// POUs/StringHelper/getCntCharInStr
{attribute 'no_check'}
//Returns the count of a particular char found in a string line
FUNCTION getCntCharInStr : INT
VAR_INPUT
	Chars													:	STRING(5):=';';
	Strline													:	T_MaxString;
END_VAR             										
VAR                 
	tmpString												:	T_MaxString ;										
	pos,k													:	INT;
END_VAR

IF StrLine <> '' AND Chars <> ''
THEN
	MEMSET(ADR(tmpString),0,SIZEOF(tmpString));
	MEMCPY(ADR(tmpString),ADR(Strline),TO_UDINT(LEN(Strline)));
	pos 													:= FIND (tmpString,Chars);
	WHILE pos <> 0 DO	
		k													:=  pos + (LEN(Chars) - 1);
		tmpString											:=	RIGHT(tmpString,LEN(tmpString) - k);
		pos 												:= 	FIND (tmpString,Chars);
		getCntCharInStr										:=	getCntCharInStr+1;
	END_WHILE;
ELSE
	getCntCharInStr											:= 0;
END_IF

END_FUNCTION

// POUs/StringHelper/getCntCharInWStr
{attribute 'no_check'}
//Returns the count of a particular char found in a string line
FUNCTION getCntCharInWStr : INT
VAR_INPUT
	Char													:	WSTRING(3):=";";
	Strline													:	WSTRING(MAX_STRING_LENGTH);
END_VAR             										
VAR                 
	tmpString												:	WSTRING(MAX_STRING_LENGTH) ;										
	pos,k													:	INT;
END_VAR

IF Strline <> "" AND Char <> ""
THEN	
	MEMSET(ADR(tmpString),0,SIZEOF(tmpString));
	MEMCPY(ADR(tmpString),ADR(Strline),TO_UDINT(WLEN(Strline) * 2));
	pos 													:= WFIND (tmpString,char);
	WHILE pos <> 0 DO		
		k													:=  pos + (WLEN(char) - 1);
		tmpString											:=	WRIGHT(tmpString,WLEN(tmpString) - k);
		pos 												:= 	WFIND (tmpString,char);
		getCntCharInWStr									:=	getCntCharInWStr+1;
	END_WHILE;
ELSE
	getCntCharInWStr										:= 0;
END_IF

END_FUNCTION

// POUs/StringHelper/getFilledString
{attribute 'no_check'}
//Returns a string which is filled with a defined char on the left or right site with a desired lenght  
FUNCTION getFilledString : T_MaxString
VAR_INPUT
	Strline													:	T_MaxString;	//Start string
	Lenght													:	INT;			//Desired lenght
	FillChar												:	STRING(1);		//Fill char
	LeftInsert												:	BOOL;			//Insert char on left site of start string
END_VAR             										
VAR                 										
	tmp														:	T_MaxString;
	i 														: INT;
END_VAR

GetFilledString 											:= Strline;
tmp 														:= '';

FOR i := 0 TO Lenght DO
	IF LEN(getFilledString)+ Lenght >= UINT_TO_INT(SIZEOF(getFilledString)) 
	THEN
		RETURN;
	ELSE
		IF LeftInsert 
		THEN
			IF LEN(tmp) < Lenght - LEN(Strline) 
			THEN
				tmp 										:= INSERT(tmp,FillChar,LEN(tmp));
			ELSE
				getFilledString 							:= CONCAT(tmp,getFilledString);
			END_IF                  						
		ELSE                        						
			getFilledString									:= INSERT(getFilledString,FillChar,LEN(getFilledString));
		END_IF
	END_IF
END_FOR

END_FUNCTION

// POUs/StringHelper/HEXSTR_TO_DWORD
{attribute 'no_check'}
//Converts a hex string into a 32 bit DWORD number
FUNCTION HEXSTR_TO_DWORD : BOOL //Return value TRUE = successful converted / FALSE if there are no valid hex signs or seperators
VAR_INPUT
	Hexstring 												: T_MaxString;
END_VAR
VAR_IN_OUT
{attribute 'displaymode':='hexadecimal'}
	Target													: DWORD;
END_VAR
VAR
	HexMarkerFound											: BOOL;
	i,j,Max_i,Max_j											: INT;
{attribute 'displaymode':='hexadecimal'}
	X														: BYTE;
{attribute 'displaymode':='hexadecimal'}
	TmpTarget												: DWORD;
END_VAR

Max_i 														:= LEN(Hexstring) - 1;
Max_j														:= SIZEOF(Target) * 2;
TmpTarget													:= 0;
HEXSTR_TO_DWORD												:= TRUE;
FOR i := 0 TO Max_i DO
	(* read the first character and subtract 48 to get value in decimal 0 = 48 *)
	(* calculate the value of the digit *)
	X														:= Hexstring[i];
	IF j >= Max_j
	THEN
		EXIT;
	ELSIF X > 47 AND x < 58 
	THEN //x = number 0-9
		TmpTarget 											:= SHL(TmpTarget,4) + X - 48;
		j													:= j + 1;
	ELSIF X > 64 AND X < 71 								
	THEN //x = letter A-F                   								
		TmpTarget 											:= SHL(TmpTarget,4) + X - 55;
		j													:= j + 1;
	ELSIF X > 96 AND X < 103								 
	THEN //x = letter a-f                     								
		TmpTarget 											:= SHL(TmpTarget,4) + X - 87;
		j													:= j + 1;
	ELSIF x = 16#58 OR x = 16#78 OR  x = 16#23
	THEN //found x, X or #, start over again because of 0xFA or 16#AB
		IF HexMarkerFound
		THEN
			HEXSTR_TO_DWORD									:= FALSE;	
			RETURN;		
		ELSE
			TmpTarget										:= 0;
			HexMarkerFound									:= TRUE;
			j												:= 0;	
		END_IF		
	ELSIF X = 16#2C OR X = 16#3A OR X = 16#2E OR X = 16#3B OR X = 16#20 OR X = 16#5F
	THEN //Ignore comma,colon,dot,space,underline
		; 
	ELSE
		HEXSTR_TO_DWORD										:= FALSE;	
		RETURN;
	END_IF
END_FOR
Target														:= TmpTarget;

END_FUNCTION

// POUs/StringHelper/HEXSTR_TO_LWORD
{attribute 'no_check'}
//Converts a hex string into a 64 bit LWORD number
FUNCTION HEXSTR_TO_LWORD : BOOL //Return value TRUE = successful converted / FALSE if there are no valid hex signs or seperators
VAR_INPUT
	Hexstring 												: T_MaxString;
END_VAR
VAR_IN_OUT
{attribute 'displaymode':='hexadecimal'}
	Target													: LWORD;
END_VAR
VAR
	HexMarkerFound											: BOOL;
	i,j,Max_i,Max_j											: INT;
{attribute 'displaymode':='hexadecimal'}
	X														: BYTE;
{attribute 'displaymode':='hexadecimal'}
	TmpTarget												: LWORD;
END_VAR

Max_i 														:= LEN(Hexstring) - 1;
Max_j														:= SIZEOF(Target) * 2;
TmpTarget 													:= 0;
HEXSTR_TO_LWORD												:= TRUE;
FOR i := 0 TO Max_i DO
	(* read the first character and subtract 48 to get value in decimal 0 = 48 *)
	(* calculate the value of the digit *)
	X														:= Hexstring[i];
	IF j >= Max_j
	THEN
		EXIT;
	ELSIF X > 47 AND x < 58 
	THEN //x = number 0-9
		TmpTarget 											:= SHL(TmpTarget,4) + X - 48;
		j													:= j + 1;
	ELSIF X > 64 AND X < 71 								
	THEN //x = letter A-F                   								
		TmpTarget 											:= SHL(TmpTarget,4) + X - 55;
		j													:= j + 1;
	ELSIF X > 96 AND X < 103								 
	THEN //x = letter a-f                     								
		TmpTarget 											:= SHL(TmpTarget,4) + X - 87;
		j													:= j + 1;
	ELSIF x = 16#58 OR x = 16#78 OR  x = 16#23
	THEN //found x, X or #, start over again because of 0xFA or 16#AB
		IF HexMarkerFound
		THEN
			HEXSTR_TO_LWORD									:= FALSE;	
			RETURN;		
		ELSE
			TmpTarget										:= 0;
			HexMarkerFound									:= TRUE;
			j												:= 0;	
		END_IF		
	ELSIF X = 16#2C OR X = 16#3A OR X = 16#2E OR X = 16#3B OR X = 16#20 OR X = 16#5F
	THEN //Ignore comma,colon,dot,space,underline
		; 
	ELSE
		HEXSTR_TO_LWORD										:= FALSE;	
		RETURN;
	END_IF
END_FOR
Target														:= TmpTarget;

END_FUNCTION

// POUs/StringHelper/isWStringNumeric
{attribute 'no_check'}
//Returns TRUE in case a ascii string contains only a valid number signs. Minus,plus,space,comma and dot are allowed
//Limited to a Param.MAX_EXT_STRING_LENGTH long string  
FUNCTION isWStringNumeric : BOOL 
VAR_INPUT
	pSource													:	POINTER TO WORD;
END_VAR             										
VAR                 
	Cr														:	WORD;	//Char									
	countSeperator											:	INT;
	i														:	UDINT;
	Addr													:	POINTER TO WORD;
END_VAR

IF pSource <> 0
THEN
	isWStringNumeric										:=	TRUE;
	FOR i := 0 TO PARAM.MAX_EXT_STRING_LENGTH DO
		Addr												:= pSource + (i * 2);
		Cr												:= Addr^;
		IF Cr = 0
		THEN 														
			isWStringNumeric								:= i > 0; //Only TRUE if string is not empty 
			EXIT;
		ELSIF Cr = 46 OR Cr = 44 //comma or point as a seperator
		THEN
			countSeperator									:= countSeperator + 1;
			IF countSeperator > 1 
			THEN
				isWStringNumeric							:= FALSE;
				EXIT;	(* more than one seperator -> no number *)
			END_IF
		ELSIF(Cr < 48 OR Cr > 57)
			AND Cr <> 45 (* minus *)
			AND Cr <> 43 (* plus *)
			AND Cr <> 32 (* Space *)
			AND Cr <> 101(* e for 9.9999992e-2 *)
			OR i = PARAM.MAX_EXT_STRING_LENGTH
		THEN
			isWStringNumeric								:= FALSE;
			EXIT;	(* no numerical char *)
		END_IF
	END_FOR      
ELSE
	isWStringNumeric										:= FALSE;
END_IF

END_FUNCTION

// POUs/StringHelper/LWORD_TO_BINSTR_EXT
{attribute 'no_check' := ''}
FUNCTION LWORD_TO_BINSTR_EXT : T_MaxString //This function converts a decimal number into a binary string (base 2), where the digits are separated according to the selected mode 
//e.g. 1111000011110000 -> 1111_0000_1111_0000 
VAR_INPUT
	In														: LWORD;//The decimal number requiring conversion.
	Precision												: INT; //Minimum number of displayed digits (digits), filled up with 0 from left if significant digits are less then that
	Mode													: INT; //1=Separate high and low word / 2=Separate bytes / 3=Separate nibbles /ELSE no separation | Separator = Param.DOWRD_TO_XXXSTR_EXT_SEPARATOR
END_VAR
VAR													
END_VAR

LWORD_TO_BINSTR_EXT 										:= LWORD_TO_BINSTR(in,precision);

CASE mode OF
1:// Separate by low word and high word
	LWORD_TO_BINSTR_EXT										:= INSERT_EXT(LWORD_TO_BINSTR_EXT,PARAM.XWORD_TO_XXXSTR_EXT_SEPARATOR,16);
	
2://Separate by bytes
	LWORD_TO_BINSTR_EXT										:= INSERT_EXT(LWORD_TO_BINSTR_EXT,PARAM.XWORD_TO_XXXSTR_EXT_SEPARATOR,8);
	
3://Separate by nibble
	LWORD_TO_BINSTR_EXT										:= INSERT_EXT(LWORD_TO_BINSTR_EXT,PARAM.XWORD_TO_XXXSTR_EXT_SEPARATOR,4);
END_CASE

END_FUNCTION

// POUs/StringHelper/LWORD_TO_HEXSTR_EXT
{attribute 'no_check' := ''}
FUNCTION LWORD_TO_HEXSTR_EXT : T_MaxString //This function converts a decimal number into a hexadecimal string (base 16)., where the hex signs are separated according to the selected mode 
//e.g. F0F0F0F0 -> F0_F0_F0_F0 
VAR_INPUT
	In														: LWORD;
	Precision												: INT;//Minimum number of displayed signs, filled up with 0 from left if significant digits are less then that
	LoCase													: BOOL;
	Mode													: INT; //1=parted by word, 2=parted by byte, 3=parted by nibble
END_VAR
VAR
END_VAR

LWORD_TO_HEXSTR_EXT 										:= LWORD_TO_HEXSTR(in,precision,loCase);
CASE mode OF
1:// Separate by low word and high word
	LWORD_TO_HEXSTR_EXT										:= INSERT_EXT(LWORD_TO_HEXSTR_EXT,PARAM.XWORD_TO_XXXSTR_EXT_SEPARATOR,4);
	
2://Separate by bytes
	LWORD_TO_HEXSTR_EXT										:= INSERT_EXT(LWORD_TO_HEXSTR_EXT,PARAM.XWORD_TO_XXXSTR_EXT_SEPARATOR,2);
	
3://Separate by nibble
	LWORD_TO_HEXSTR_EXT										:= INSERT_EXT(LWORD_TO_HEXSTR_EXT,PARAM.XWORD_TO_XXXSTR_EXT_SEPARATOR,1);
END_CASE

END_FUNCTION

// POUs/StringHelper/readWStrToSeperator
{attribute 'no_check'}
//Returns a wstring found on the left side of a seperator, empty if seperator is not found
FUNCTION readWStrToSeperator : WSTRING(MAX_STRING_LENGTH)
VAR_INPUT
	Seperator												:	WSTRING(10) :=";";
	Strline													:	WSTRING(MAX_STRING_LENGTH);
END_VAR
VAR_IN_OUT
END_VAR
VAR
	pos														:	INT;
END_VAR

IF strline = ""
THEN
	readWStrToSeperator										:= "";
ELSE
	pos 													:= WFIND (strline,seperator);
	IF (pos >= 1) 
	THEN
		readWStrToSeperator									:= WLEFT (strline,pos-1);
	ELSE
		readWStrToSeperator									:= "";
	END_IF
END_IF

END_FUNCTION

// POUs/StringHelper/replaceInString
{attribute 'no_check'}
//Replace a part of a string with another string 
FUNCTION replaceInString : BOOL
VAR_INPUT
	SearchStr												:	STRING(10); //e.g. '/r/n_
	ReplaceStr												:	STRING(10); //e.g. '-'
END_VAR             										
VAR_IN_OUT         										
	Strline													: 	T_MaxString;
END_VAR             										
VAR                 	
	StrLen, i,pos											:	INT;
END_VAR

IF strline = '' 
THEN 
	replaceInString											:= TRUE;
ELSE
	StrLen													:= LEN(strline);
	FOR i := 0 TO StrLen
	DO
		pos 												:= FIND(strline,SearchStr);
		IF pos >= 1 
		THEN
			strline											:= REPLACE(strline,ReplaceStr,LEN(SearchStr),pos);
		ELSE
			replaceInString									:= i > 0; 
			EXIT;						
		END_IF	
	END_FOR
END_IF

END_FUNCTION

// POUs/StringHelper/replaceInWString
{attribute 'no_check'}
//Replace a part of a string with another string 
FUNCTION replaceInWString : BOOL
VAR_INPUT
	SearchStr												:	WSTRING(10); //e.g. '/r/n_
	ReplaceStr												:	WSTRING(10); //e.g. '-'
END_VAR             										
VAR_IN_OUT         										
	Strline													: 	WSTRING(MAX_STRING_LENGTH);
END_VAR             										
VAR                 	
	StrLen, i,pos											:	INT;
END_VAR

IF strline = "" 
THEN 
	replaceInWString										:= TRUE;
ELSE
	StrLen													:= WLEN(strline);
	FOR i := 0 TO StrLen
	DO
		pos 												:= WFIND(strline,SearchStr);
		IF pos >= 1 
		THEN
			strline											:= WREPLACE(strline,ReplaceStr,WLEN(SearchStr),pos);
		ELSE
			replaceInWString								:= i > 0; 
			EXIT;						
		END_IF	
	END_FOR
END_IF

END_FUNCTION

// POUs/StringHelper/replaceUmlauts
// ReplaceUmlauts replaces all "german" umlauts in an given string Ä-> ae | ä -> ae | Ö -> oe | ö -> oe | Ü -> ue | ü -> ue | ß -> ss 
FUNCTION replaceUmlauts : INT // returns no of replaced umlauts
VAR_IN_OUT
	SearchStr		: T_MaxString;				
END_VAR
VAR
	i			: INT;
END_VAR

FOR i := 0 TO LEN(SearchStr) DO
	CASE SearchStr[i] OF
	196:	// Ä
		SearchStr 					:= REPLACE(SearchStr, 'Ae', 1, i+1); 
		i 							:= i + 1;
		ReplaceUmlauts 				:= ReplaceUmlauts + 1;
	214:	// Ö
		SearchStr 					:= REPLACE(SearchStr, 'Oe', 1, i+1);
		i 							:= i + 1; 
		ReplaceUmlauts 				:= ReplaceUmlauts + 1;
	220:	// Ü
		SearchStr 					:= REPLACE(SearchStr, 'Ue', 1, i+1);
		i 							:= i + 1; 
		ReplaceUmlauts 				:= ReplaceUmlauts + 1;
	223:	// ß
		SearchStr 					:= REPLACE(SearchStr, 'ss', 1, i+1);
		i 							:= i + 1; 
		ReplaceUmlauts 				:= ReplaceUmlauts + 1;	
	228:	// ä
		SearchStr 					:= REPLACE(SearchStr, 'ae', 1, i+1);
		i 							:= i + 1; 
		ReplaceUmlauts 				:= ReplaceUmlauts + 1;
	246:	// ö
		SearchStr 					:= REPLACE(SearchStr, 'oe', 1, i+1);
		i 							:= i + 1; 
		ReplaceUmlauts 				:= ReplaceUmlauts + 1;
	252:	// ü
		SearchStr 					:= REPLACE(SearchStr, 'ue', 1, i+1);
		i 							:= i + 1; 
		ReplaceUmlauts 				:= ReplaceUmlauts + 1;
	ELSE	// nothing replaced in this cycle	
		;
	END_CASE
END_FOR

END_FUNCTION

// POUs/StringHelper/WINSERT_EXT
{attribute 'no_check' := ''}
FUNCTION WINSERT_EXT : WSTRING //The function WINSERT_EXT inserts WSTR2 into WSTR1 at every ITERATION_POSs position  
VAR_INPUT
	STR1													:WSTRING; //Base string - Hint! The base string will cut off if iteration of insertions exceeded the size of the string variable 
	STR2													:WSTRING; //Insert string 
	ITERATION_POS											: INT; //Insert iteration position 
END_VAR
VAR
	Length1,length2,i,iEnd									: INT;														
END_VAR

WINSERT_EXT													:= STR1;
Length1														:= WLEN(STR1);
Length2														:= WLEN(STR2);
IF TO_UINT(Length1 + Length2) > SIZEOF(STR1)
	OR ITERATION_POS = 0
THEN
	;
ELSE
	iEnd													:= ABS(Length1 / ITERATION_POS) - 1;
	FOR i := 1 TO iEnd
	DO 
		WINSERT_EXT											:= WINSERT(WINSERT_EXT,STR2,Length1 - ITERATION_POS * i);
	END_FOR
END_IF

END_FUNCTION

// POUs/System/SystemPulses
{attribute 'no_check'}
//Provides various puslse signals as default
FUNCTION_BLOCK SystemPulses
VAR_INPUT
{attribute 'displaymode':='binary'}
	Options													:	WORD := 2#0000_0001_1110_1110; //Set bit in Options word to enable ot disable existing pulse instances
	PT_ON_Custom											:	TIME := T#30S;	
	PT_OFF_Custom											:	TIME := T#30S;
END_VAR
VAR_OUTPUT
	BlinkSlow												: 	BOOL;
	Blink													: 	BOOL;
	BlinkFast												: 	BOOL;
	BlinkVeryFast											:	BOOL;
	BlinkFlash												:	BOOL;
	
	_20ms													: 	Pulse := (IN := TRUE,	PT_OFF := T#20MS, 		PT_ON := T#20MS);	//20ms						Options .0
	_100ms													: 	Pulse := (IN := TRUE,	PT_OFF := T#100MS, 		PT_ON := T#100MS); 	//10Hz (0.1s) pulse			Options .1
	_250ms													: 	Pulse := (IN := TRUE,	PT_OFF := T#250MS, 		PT_ON := T#250MS); 	//4 Hz - Blink very Fast	Options .2
	_400ms													: 	Pulse := (IN := TRUE,	PT_OFF := T#400MS, 		PT_ON := T#400MS); 	//2.5Hz - Blink Fast *)		Options .3
	_500ms													: 	Pulse := (IN := TRUE,	PT_OFF := T#500MS, 		PT_ON := T#500MS); 	//2Hz / 500ms				Options .4
	_800ms													: 	Pulse := (IN := TRUE,	PT_OFF := T#800MS, 		PT_ON := T#800MS); 	//1.25Hz - Blink normal 	Options .5
	_1s														: 	Pulse := (IN := TRUE,	PT_OFF := T#1S, 		PT_ON := T#1S); 	//1Hz /1s					Options .6
	_1s600ms												: 	Pulse := (IN := TRUE,	PT_OFF := T#1S600MS, 	PT_ON := T#1S600MS);//0.625Hz - Blink slow 		Options .7
	_2s														: 	Pulse := (IN := TRUE,	PT_OFF := T#2S, 		PT_ON := T#2S); 	//0.5Hz						Options .8
	_5s														: 	Pulse := (IN := TRUE,	PT_OFF := T#5S, 		PT_ON := T#5S); 	//5s						Options .9
	_10s													: 	Pulse := (IN := TRUE, 	PT_OFF := T#10S, 		PT_ON := T#10S); 	//10s						Options .10
	_1m														: 	Pulse := (IN := TRUE, 	PT_OFF := T#1M, 		PT_ON := T#1M); 	//1m						Options .11	
	_5m														: 	Pulse := (IN := TRUE, 	PT_OFF := T#5M, 		PT_ON := T#5M); 	//5m						Options .12
	_10m													: 	Pulse := (IN := TRUE, 	PT_OFF := T#10M, 		PT_ON := T#10M); 	//10m						Options .13
	_60m													: 	Pulse := (IN := TRUE, 	PT_OFF := T#60M, 		PT_ON := T#60M); 	//60m						Options .14
	_Custom													: 	Pulse := (IN := TRUE, 	PT_OFF := T#30S, 		PT_ON := T#60M); 	//60m						Options .15
	_Flash													: 	Pulse := (IN := TRUE, 	PT_OFF := T#800MS, 		PT_ON := T#80MS);	//800ms/80ms Blink as flash light
END_VAR                                                            
VAR                                                                
END_VAR

(************************************************************************************************************)
(* function-block generates different pulse signals															*)
(************************************************************************************************************)

(* impuls generator *****************************************************************************************)
_Flash(Q => BlinkFlash); 
IF Options.0 THEN _20ms(Q => ); 				END_IF
IF Options.1 THEN _100ms(Q => ); 				END_IF
IF Options.2 THEN _250ms(Q => BlinkVeryFast); 	END_IF
IF Options.3 THEN _400ms(Q => BlinkFast); 		END_IF
IF Options.4 THEN _500ms(Q => ); 				END_IF
IF Options.5 THEN _800ms(Q => Blink); 			END_IF
IF Options.6 THEN _1s(Q => ); 					END_IF
IF Options.7 THEN _1s600ms(Q => BlinkSlow); 	END_IF
IF Options.8 THEN _2s(Q => ); 					END_IF
IF Options.9 THEN _5s(Q => ); 					END_IF
IF Options.10 THEN _10s(Q => ); 				END_IF
IF Options.11 THEN _1m(Q => ); 					END_IF
IF Options.12 THEN _5m(Q => ); 					END_IF
IF Options.13 THEN _10m(Q => ); 				END_IF
IF Options.14 THEN _60m(Q => ); 				END_IF
IF Options.15 THEN _Custom(PT_OFF := PT_OFF_Custom, PT_ON := PT_ON_Custom ,Q => );	END_IF

(************************************************************************************************)

PROPERTY PUBLIC optAllOn : bool
GET
optAllOn := OPtions = 2#1111_1111_1111_1111;
END_GET
SET
If optAllOn then OPtions := 2#1111_1111_1111_1111; End_if
END_SET
END_PROPERTY

PROPERTY PUBLIC optEnable100ms : bool
GET
optEnable100ms := Options.0;
END_GET
SET
Options.0 := optEnable100ms;
END_SET
END_PROPERTY

PROPERTY PUBLIC optEnable10m : bool
GET
optEnable10m := Options.13;
END_GET
SET
Options.13 := optEnable10m;
END_SET
END_PROPERTY

PROPERTY PUBLIC optEnable10s : bool
GET
optEnable10s := Options.10;
END_GET
SET
Options.10 := optEnable10s;
END_SET
END_PROPERTY

PROPERTY PUBLIC optEnable1m : bool
GET
optEnable1m := Options.11;
END_GET
SET
Options.11 := optEnable1m;
END_SET
END_PROPERTY

PROPERTY PUBLIC optEnable1s : bool
GET
optEnable1s := Options.6;
END_GET
SET
Options.6 := optEnable1s;
END_SET
END_PROPERTY

PROPERTY PUBLIC optEnable1s600msBlinkSlow : bool
GET
optEnable1s600msBlinkSlow := Options.7;
END_GET
SET
Options.7 := optEnable1s600msBlinkSlow;
END_SET
END_PROPERTY

PROPERTY PUBLIC optEnable20ms : bool
GET
optEnable20ms := Options.0;
END_GET
SET
Options.0 := optEnable20ms;
END_SET
END_PROPERTY

PROPERTY PUBLIC optEnable250msBlinkVeryFast : bool
GET
optEnable250msBlinkVeryFast := Options.2;
END_GET
SET
Options.2 := optEnable250msBlinkVeryFast;
END_SET
END_PROPERTY

PROPERTY PUBLIC optEnable2s : bool
GET
optEnable2s := Options.8;
END_GET
SET
Options.8 := optEnable2s;
END_SET
END_PROPERTY

PROPERTY PUBLIC optEnable400msBlinkFast : bool
GET
optEnable400msBlinkFast := Options.3;
END_GET
SET
Options.3 := optEnable400msBlinkFast;
END_SET
END_PROPERTY

PROPERTY PUBLIC optEnable500ms : bool
GET
optEnable500ms := Options.4;
END_GET
SET
Options.4 := optEnable500ms;
END_SET
END_PROPERTY

PROPERTY PUBLIC optEnable5m : bool
GET
optEnable5m := Options.12;
END_GET
SET
Options.12 := optEnable5m;
END_SET
END_PROPERTY

PROPERTY PUBLIC optEnable5s : bool
GET
optEnable5s := Options.9;
END_GET
SET
Options.9 := optEnable5s;
END_SET
END_PROPERTY

PROPERTY PUBLIC optEnable60m : bool
GET
optEnable60m := Options.14;
END_GET
SET
Options.14 := optEnable60m;
END_SET
END_PROPERTY

PROPERTY PUBLIC optEnable800msBlink : bool
GET
optEnable800msBlink := Options.5;
END_GET
SET
Options.5 := optEnable800msBlink;
END_SET
END_PROPERTY

PROPERTY PUBLIC optEnableCustom : bool
GET
optEnableCustom:= Options.15;
END_GET
SET
Options.15 := optEnableCustom;
END_SET
END_PROPERTY

END_FUNCTION_BLOCK

// POUs/System/TaskInfo
{attribute 'no_check'}
//Provides all information of PlcTaskSystemInfo corresponding to the caller task of the instance 
FUNCTION_BLOCK TaskInfo
VAR_INPUT
END_VAR
VAR_OUTPUT
	Index													:	INT := 0;
	TaskName          										: 	STRING(63);
	ObjId             										: 	OTCID;
	CycleTime         										: 	UDINT;
	CycleTimeT       										: 	TIME;
	CycleTimeLT       										: 	LTIME;
	CycleTimeFloat											:	LREAL;	
	Priority          										: 	UINT;
	AdsPort           										: 	UINT;
	CycleCount        										: 	UDINT;
	Tasktime												:	ULINT;
	DcTaskTime        										: 	T_DCTIME64;
	LastExecTime      										: 	UDINT; 
	LastExecTimeNS      									: 	UDINT; //Converted in ns 
	LastExecTimeLT      									: 	LTIME; 
	MaxExecTimeLT											:	LTIME;
	FirstCycle        										: 	BOOL;
	CycleTimeExceeded 										: 	BOOL;	
	CycleTimeExceededCount 									: 	UDINT; //Set to 0 via method resetCylceTimeExceeded()
	CycleTimeExceededCountTotal 							: 	UDINT; //Overall count cycle time exeeded
	InCallAfterOutputUpdate									:	BOOL;
	RTViolation												:	BOOL;
END_VAR

VAR
	GETCURTASKINDEX											: 	GETCURTASKINDEX;
	GETTASKTIME												:	GETTASKTIME;
	TaskInterlock											:	BOOL;
END_VAR

	(*	evaluate PlcTaskInfo arrays													*)
	(********************************************************************************)

(* read task info array of caller task ************************************************************************)
	IF GETCURTASKINDEX.index = 0 	
	THEN 
		GETCURTASKINDEX(index => index); 
		//Init
		TaskName          									:= TwinCAT_SystemInfoVarList._TaskInfo[index].TaskName;
		ObjId             									:= TwinCAT_SystemInfoVarList._TaskInfo[index].ObjId;
		CycleTime         									:= TwinCAT_SystemInfoVarList._TaskInfo[index].CycleTime;
		Priority          									:= TwinCAT_SystemInfoVarList._TaskInfo[index].Priority;
		AdsPort           									:= TwinCAT_SystemInfoVarList._TaskInfo[index].AdsPort;
		CycleTimeT											:= LREAL_TO_TIME(UDINT_TO_LREAL(CycleTime) * 0.0001 );
		CycleTimeLT											:= TO_LTIME(CycleTime * 100);
		CycleTimeFloat										:= (UDINT_TO_LREAL(CycleTime) * 0.0001 / 1000.0);		
	END_IF

	//Cylic 
	CycleCount        										:= TwinCAT_SystemInfoVarList._TaskInfo[index].CycleCount;
	DcTaskTime        										:= TO_ULINT(TwinCAT_SystemInfoVarList._TaskInfo[index].DcTaskTime); 
	LastExecTime      										:= TwinCAT_SystemInfoVarList._TaskInfo[index].LastExecTime; 
	LastExecTimeNS											:= TwinCAT_SystemInfoVarList._TaskInfo[index].LastExecTime * 100;
	LastExecTimeLT      									:= TO_LTIME(LastExecTimeNS); //Converted into ns 
	MaxExecTimeLT											:= MAX(LastExecTimeLT,MaxExecTimeLT);
	
	FirstCycle        										:= TwinCAT_SystemInfoVarList._TaskInfo[index].FirstCycle;
	CycleTimeExceeded 										:= TwinCAT_SystemInfoVarList._TaskInfo[index].CycleTimeExceeded;
	IF CycleTimeExceeded 
	THEN
		CycleTimeExceededCount								:= CycleTimeExceededCount + 1;	
		CycleTimeExceededCountTotal							:= CycleTimeExceededCountTotal + 1;
	END_IF
	InCallAfterOutputUpdate									:= TwinCAT_SystemInfoVarList._TaskInfo[index].InCallAfterOutputUpdate;
	RTViolation												:= TwinCAT_SystemInfoVarList._TaskInfo[index].RTViolation;
	
	//Read time when task suppose to start
	GETTASKTIME(timeLoDW => Tasktime);	
	MEMCPY(ADR(Tasktime) + SIZEOF(GETTASKTIME.timeHiDW),ADR(GETTASKTIME.timeHiDW),SIZEOF(GETTASKTIME.timeHiDW));
	
(**************************************************************************************************)

METHOD PUBLIC resetCylceTimeExceeded : BOOL //Return value = TRUE if execution finished
VAR_INPUT
END_VAR
IF TestAndSet(TaskInterlock)
THEN
	CycleTimeExceededCount									:= 0;
	TaskInterlock											:= FALSE;
	resetCylceTimeExceeded											:= TRUE;
END_IF
END_METHOD

END_FUNCTION_BLOCK

// POUs/TimeHelper/Conversions/FILETIME_TO_DATE
FUNCTION FILETIME_TO_DATE : DATE //Converts 64bit T_FILETIME to DATE (D#1970-01-01)
VAR_INPUT
	IN														: T_FILETIME;
END_VAR
VAR
END_VAR

FILETIME_TO_DATE											:= DT_TO_DATE(FILETIME_TO_DT(IN));

END_FUNCTION

// POUs/TimeHelper/Conversions/FILETIME_TO_TOD
FUNCTION FILETIME_TO_TOD : TIME_OF_DAY //Converts 64bit T_FILETIME to TIME_OF_DAY (TOD#15:36:30.123)
VAR_INPUT
	IN														: T_FILETIME;
END_VAR
VAR
END_VAR

FILETIME_TO_TOD												:= SYSTEMTIME_TO_TOD(FILETIME_TO_SYSTEMTIME(IN));

END_FUNCTION

// POUs/TimeHelper/Conversions/SYSTEMTIME_TO_TOD
FUNCTION SYSTEMTIME_TO_TOD : TIME_OF_DAY //Converts Systemtime (Timestruct) to TIME_OF_DAY (TOD#15:36:30.123)
VAR_INPUT
	IN													: TIMESTRUCT;
END_VAR
VAR
END_VAR

SYSTEMTIME_TO_TOD											:= UDINT_TO_TOD(IN.wMilliseconds 
																+ IN.wSecond * 1000
																+ IN.wMinute * 60000
																+ IN.wHour * 3600000);

END_FUNCTION

// POUs/TimeHelper/Conversions/LREAL_TO_TIME_SEC
{attribute 'no_check'}
//Convert time in lreal format <s.ms> into time format 
FUNCTION LREAL_TO_TIME_SEC : TIME
VAR_INPUT
	 IN														: LREAL;
END_VAR
VAR
END_VAR

LREAL_TO_TIME_SEC 											:= LREAL_TO_TIME(IN * 1000.0);

END_FUNCTION

// POUs/TimeHelper/Conversions/SYSTEMTIME_TO_DATE
FUNCTION SYSTEMTIME_TO_DATE : DATE //Converts Systemtime (Timestruct) to DATE (D#2020-06-02)
VAR_INPUT
	IN													: TIMESTRUCT;
END_VAR
VAR
END_VAR

SYSTEMTIME_TO_DATE										:= DT_TO_DATE(SYSTEMTIME_TO_DT(IN));

END_FUNCTION

// POUs/TimeHelper/Conversions/SYSTEMTIME_TO_TIME
FUNCTION SYSTEMTIME_TO_TIME : TIME //Converts Systemtime (Timestruct) of day to TIME (T#15h23m12s34ms)
VAR_INPUT
	IN													: TIMESTRUCT;
END_VAR
VAR
END_VAR

SYSTEMTIME_TO_TIME											:= TO_TIME(IN.wMilliseconds
																+ IN.wSecond * 1000
																+ IN.wMinute * 60000
																+ IN.wHour * 3600000);

END_FUNCTION

// POUs/TimeHelper/Conversions/SYSTEMTIME_TO_TIME_EX
FUNCTION SYSTEMTIME_TO_TIME_EX : TIME //Converts Systemtime (Timestruct) to TIME incl. day of week (T#3d15h23m12s34ms), which means the value reflects the time of the week starting from Sunday (DayOfWeek=0) 
VAR_INPUT
	IN													: TIMESTRUCT;
END_VAR
VAR
END_VAR

SYSTEMTIME_TO_TIME_EX											:= TO_TIME(IN.wMilliseconds 
																+ IN.wSecond * 1000
																+ IN.wMinute * 60000
																+ IN.wHour * 3600000
																+ IN.wDayOfWeek * 86400000);

END_FUNCTION

// POUs/TimeHelper/Conversions/TIME_TO_FMRLREAL
{attribute 'no_check'}
//Convert a time value into a Lreal value in <s.ms> 
FUNCTION TIME_TO_FMRLREAL : LREAL
VAR_INPUT
	TIME_IN													:	TIME;
	NoOfDigits												:   INT(0..10) := 0; (* amount of decimaldigis*)
END_VAR             										
VAR                     									
	X														:	LREAL;
END_VAR

TIME_TO_FMRLREAL 											:= TIME_TO_LREAL(TIME_IN) ;
IF NoOfDigits > 0
THEN
	X														:= EXPT(10.0,ABS( NoOfDigits));
	TIME_TO_FMRLREAL										:= TIME_TO_FMRLREAL / X;
END_IF

END_FUNCTION

// POUs/TimeHelper/Conversions/TIME_TO_SYSTEMTIME
FUNCTION TIME_TO_SYSTEMTIME : TIMESTRUCT //Converts Systemtime (Timestruct) of day to TIME (T#15h23m12s34ms)
VAR_INPUT
	IN														: TIME;
END_VAR
VAR
	n														:	UDINT;
END_VAR

n															:= TO_UDINT(IN);
TIME_TO_SYSTEMTIME.wDayOfweek								:= TO_WORD(n / 86400000);
n															:= n - (TIME_TO_SYSTEMTIME.wDayOfweek * 86400000);
														
TIME_TO_SYSTEMTIME.wHour									:= TO_WORD(n / 3600000);
n															:= n - (TIME_TO_SYSTEMTIME.wHour * 3600000);

TIME_TO_SYSTEMTIME.wMinute									:= TO_WORD(n / 60000);
n															:= n - (TIME_TO_SYSTEMTIME.wMinute * 60000);

TIME_TO_SYSTEMTIME.wSecond									:= TO_WORD(n / 1000);
n															:= n - (TIME_TO_SYSTEMTIME.wSecond * 1000);

TIME_TO_SYSTEMTIME.wMilliseconds							:= TO_WORD(n);	

TIME_TO_SYSTEMTIME.wDay										:= 0;
TIME_TO_SYSTEMTIME.wYear									:= 0;
TIME_TO_SYSTEMTIME.wMonth									:= 0;

END_FUNCTION

// POUs/TimeHelper/createTOD
{attribute 'no_check'}
//Creates a TOD value based on the input parameter
FUNCTION createTOD : TOD
VAR_INPUT
   Hour            											: WORD;
   Minute          											: WORD;
   Second          											: WORD;
   Milliseconds    											: WORD;
END_VAR
VAR
	X														:	UDINT;
END_VAR

createTOD 													:= UDINT_TO_TOD(	Milliseconds 
																				+ (Second * 1000)
																				+ (Minute * 60000)
																				+ (Hour * 3600000));

END_FUNCTION

// POUs/TimeHelper/getDateAndTimeDelta
{attribute 'no_check'}
//calcualte the difference between two DATE_AND_TIME variables
FUNCTION getDateAndTimeDelta : TIMESTRUCT
VAR_INPUT
	IN1														: DATE_AND_TIME;
	IN2														: DATE_AND_TIME;
END_VAR             										
VAR                 										
	diff													:	DWORD;
	Result													:	TIMESTRUCT;
END_VAR

IF IN1 > IN2 
THEN
	diff 													:= DT_TO_DWORD(IN1) - DT_TO_DWORD(IN2);
	Result 													:= DT_TO_SYSTEMTIME(DWORD_TO_DT(diff));
	Result.wYear											:= Result.wYear - 1970;
	Result.wDay 											:= Result.wDay - 1;
	Result.wDayOfWeek 										:= 0;
	Result.wMonth 											:= Result.wMonth - 1;
ELSIF IN1 < IN2 
THEN
	diff 													:= DT_TO_DWORD(IN2) - DT_TO_DWORD(IN1);
	Result 													:= DT_TO_SYSTEMTIME(DWORD_TO_DT(diff));
	Result.wYear 											:= Result.wYear - 1970;
	Result.wDay 											:= Result.wDay - 1;
	Result.wDayOfWeek 										:= 0;
	Result.wMonth 											:= Result.wMonth - 1;
ELSE
	MEMSET(ADR(Result),0,SIZEOF(Result));
END_IF
getDateAndTimeDelta 										:= Result;

END_FUNCTION

// POUs/TimeHelper/getTonCountdown
{attribute 'no_check'}
//Provides the countdown value of an TON timer
FUNCTION getTonCountdown : TIME
VAR_IN_OUT
	Timer													:	TON;
END_VAR
VAR
END_VAR

IF Timer.IN
	AND NOT Timer.Q
THEN
	getTonCountdown 										:= Timer.PT - Timer.ET;
ELSE
	getTonCountdown 										:= T#0MS;
END_IF

END_FUNCTION

// POUs/TimeHelper/LivebitCheck
{attribute 'no_check'}
//Livebit monitoring
FUNCTION_BLOCK LivebitCheck
VAR_INPUT
	IN														: 	BOOL := FALSE;//Livebit signal
	RST														:	BOOL := TRUE; //Reset error output Q
	PT														: 	TIME := T#5S; //Livebit timeout
END_VAR     												
VAR_OUTPUT  												
	Q														: 	BOOL := FALSE; //True if livebit is stable for longer then PT time
END_VAR
VAR
	TON_TO 													: TON;
	M														:	BOOL;
END_VAR

(* watches the livebit toggle														*)
(************************************************************************************)

(* process ***************************************************************************)
TON_TO(IN := (IN XOR NOT M), PT := PT);
M 															:= IN;
Q 															:= TON_TO.Q OR (Q AND NOT RST);

(************************************************************************************)

END_FUNCTION_BLOCK

// POUs/TimeHelper/Ontime
{attribute 'no_check'}
//Ontime with retain outputs - Attention, if the FB will be declared inside a FB or PRG poe, the whole poe will be part of the retain data too
FUNCTION_BLOCK Ontime
VAR_INPUT
	IN 														: 	BOOL	:= FALSE;	//Start ontime counter
	ReseTrig 												: 	BOOL	:= FALSE;	//Reset counter values
END_VAR
VAR_OUTPUT
	MinAtThisCycle											:	UDINT;			//Ontime at current cycle in minutes
END_VAR
VAR_OUTPUT RETAIN 
	Hours													:	UDINT;			//Recorded and accumulated total ontime in hours
	Minutes													:	UDINT;			//Recorded and accumulated total ontime in minutes
	Seconds													: 	UDINT;			//Recorded ontime in seconds
	Cycles													: 	UDINT;			//Recorded and accumulated total start cycles 
	PersistentSec											:	UDINT;			//Recorded and accumulated total ontime in seconds - not resetable
END_VAR
VAR
	txSys													: 	TIME;
	tx														:	DWORD;
	last 													: 	DWORD;
	ms														: 	DWORD;
	edge 													: 	BOOL := FALSE;
	init													:	BOOL := FALSE;
END_VAR

(* read system time *)
txSys 														:= TIME();
tx 															:= TIME_TO_DWORD(txSys);

(* make sure the first cycle works correctly *)
IF Resetrig 
THEN
	reset();
ELSIF NOT init 
THEN
	init 													:= TRUE;
	last 													:= tx;
	ms 														:= 0;
	edge													:= FALSE;
ELSIF IN 
THEN
	(* add the current milliseconds *)
	ms 														:= (tx - last) + ms;
	IF ms >= 1000 
	THEN
		Seconds 											:= Seconds + 1;
		PersistentSec										:= PersistentSec + 1;
		ms 													:= ms - 1000;
		IF Seconds >= 60 
		THEN
			Minutes											:= Minutes + 1;
			MinAtThisCycle									:= MinAtThisCycle + 1;
			Seconds											:= 0;
			IF Minutes >= 60
			THEN
				Hours										:= Hours + 1;
				Minutes										:= 0;
			END_IF
		END_IF	 
	END_IF;
	cycles 													:= cycles + BOOL_TO_UDINT(NOT edge);
ELSE
	MinAtThisCycle											:= 0;
END_IF;

edge														:= IN;
last 														:= tx;

METHOD PUBLIC reset : BOOL //Return value = TRUE if execution finished
VAR_INPUT
END_VAR
	last 													:= tx;
	ms 														:= 0;
	tx														:= 0;
	(* add the current milliseconds *)
	ms 														:= (tx - last) + ms;
	MinAtThisCycle											:= 0;
	Hours													:= 0;
	Minutes													:= 0;
	Seconds													:= 0;
	Cycles													:= 0;
	
	reset													:= TRUE;
END_METHOD

END_FUNCTION_BLOCK

// POUs/TimeHelper/OntimeExt
{attribute 'no_check'}
//Ontime function with external counter variables via references 
FUNCTION_BLOCK OntimeExt
VAR_INPUT
	IN														: 	BOOL := FALSE;		//Start ontime counting 
	ResetTrig												: 	BOOL := FALSE;		//Reset all counter
	rHour													:	REFERENCE TO UDINT;	//Ontime counter of total houres
	rMinute													:	REFERENCE TO UDINT;	//Ontime counter of minutes until one hour expired
	rSecond													:	REFERENCE TO UDINT; //Ontime counter of seconds until one minute expired
END_VAR
VAR_OUTPUT
	Error													:	BOOL;				//Invalid input references 
END_VAR
VAR
	txSys													: 	TIME;
	tx														: 	DWORD := 0;
	last													: 	DWORD := 0;
	ms														:	DWORD := 0;
	Init													:	BOOL := FALSE;
END_VAR

IF NOT __ISVALIDREF(rHour)
	OR NOT __ISVALIDREF(rMinute)
	OR NOT __ISVALIDREF(rSecond)
THEN
	Error													:= TRUE;
	RETURN;                 								
ELSE                        									
	Error 													:= FALSE;
END_IF                      	

(* read system time *)
txSys 														:= TIME();
tx 															:= TIME_TO_DWORD(txSys);
        													
(* make sure the first cycle works correctly *)
IF ResetTrig 
THEN
	reset();
ELSIF IN 
	AND Init 
THEN
	(* add the current milliseconds *)
	ms 														:= (tx - last) + ms;
	IF ms >= 1000 
	THEN
		rSecond 											:= rSecond + 1;
		IF rSecond >= 60
		THEN
			rSecond											:= 0;
			rMinute											:= rMinute + 1;
			IF rMinute >= 60
			THEN
				rMinute										:= 0;
				rHour										:= rHour + 1;
			END_IF
	  	END_IF
		ms 													:= ABS(ms - 1000);
	END_IF;
ELSE
	;
END_IF

Init 														:= TRUE;
last 														:= tx;

METHOD PUBLIC reset : BOOL //Return value = TRUE if execution finished
VAR_INPUT
END_VAR
	last 													:= tx;
	rHour 													:= rMinute := rSecond := 0;
	reset													:= TRUE;
END_METHOD

END_FUNCTION_BLOCK

// POUs/TimeHelper/OntimeSimple
{attribute 'no_check'}
//Simple ontime function, FB is not persistent as default and output as LTIME is limited to :LTIME#1000d15h23m12s34ms2us44ns
FUNCTION_BLOCK OntimeSimple
VAR_INPUT
	IN 														: BOOL	:= FALSE;
	ResetTrig 													: BOOL	:= FALSE;
END_VAR         											
VAR_OUTPUT      											
	Q														: LTIME;
END_VAR         											
VAR             											
	txSys													: 	TIME;
	tx														:	DWORD;
	last 													: 	DWORD;
END_VAR

(* read system time *)
txSys 														:= TIME();
tx 															:= TIME_TO_DWORD(txSys);

(* make sure the first cycle works correctly *)
IF ResetTrig 
THEN
	reset();
ELSIF IN 
THEN
	(* add the current milliseconds *)
	Q		 												:= TO_LTIME(tx - last)*1000000 + Q; //convert time ms to ns of LTIME
ELSE
	;
END_IF;

last 														:= tx;

METHOD PUBLIC reset : BOOL //Return value = TRUE if execution finished
VAR_INPUT
END_VAR
	Q	 													:= LTIME#0MS;
	last 													:= tx;
	reset													:= TRUE;
END_METHOD

END_FUNCTION_BLOCK

// POUs/TimeHelper/PartsPerTime
{attribute 'no_check'}
//This function-block counts pieces/parts per selectable basetime 
FUNCTION_BLOCK PartsPerTime
VAR_INPUT
	NewPartTrig												: 	BOOL	:= FALSE;	// event
	ResetTrig												: 	BOOL	:= FALSE;	// reset counter
	Basetime												:	TIME 	:= T#60S;	// basetime
END_VAR             										
VAR_OUTPUT          										
	Forecast												: 	LREAL;				// calulated forecast for basetime
	Counted													: 	DINT;				// counted impulses in last basetime period
	CountAct												:	DINT;				// actual counter in basetime period
	Q_RT													:	BOOL;				// rising event of trigger input
END_VAR             										
VAR                 										
	rtTrigger												: 	R_TRIG;
	TON														:	TON;
	StartTime												: 	TIME;
	StartTime_Old											: 	TIME;
	TimeImpImp												: 	TIME;
END_VAR

rtTrigger(CLK := NewPartTrig,Q => Q_RT);
TON(IN := NOT TON.Q AND NOT ResetTrig, PT := Basetime);

IF TON.Q 
THEN
	Counted 												:= CountAct;
	CountAct 												:= 0;
END_IF

IF ResetTrig 
THEN
	reset();
ELSIF rtTrigger.Q 
THEN
	addNewPart();
END_IF

METHOD PUBLIC addNewPart : BOOL //Return value = TRUE if execution finished
VAR_INPUT
END_VAR
	StartTime_Old 											:= StartTime;
	StartTime 												:= TIME();
	TimeImpImp	 											:= MAX(T#1MS ,StartTime - StartTime_Old);
	Forecast	 											:= 1000.0 / (TIME_TO_LREAL(TimeImpImp));
	Forecast 												:= Forecast * (TIME_TO_REAL(Basetime) * 0.001);
	CountAct 												:= CountAct + 1;
	addNewPart												:= TRUE;
	Q_RT													:= TRUE;
END_METHOD

METHOD PUBLIC reset : bool //Return value = TRUE if execution finished
VAR_INPUT
END_VAR
	Forecast												:= 0;
	Counted													:= 0;
	CountAct												:= 0;
	reset													:= TRUE;
END_METHOD

END_FUNCTION_BLOCK

// POUs/TimeHelper/SensorTimeoutCheck
{attribute 'no_check'}
//This function-block checks wheter a sensor ("IN") is to long or to short occupied, based on the values of time and velocity which are related to the lenght
//Used to detect jamped pieces on a conveyor or flickering sensors
FUNCTION_BLOCK SensorTimeoutCheck
VAR_INPUT
	Enable													:	BOOL := TRUE;	//Enable 
	In														: 	BOOL := FALSE;	//Sensor signal 
	ResetTrig												:	BOOL := FALSE;	//Ack an error
	Offset_msec												: 	TIME := T#0MS; //ms
	Offset_mm												: 	LREAL := 300.0; //mm
	LenghtMin												:	LREAL := 100.0; //mm
 	LenghtMax												:	LREAL := 1000.0; //mm
	Velo													:	LREAL := 1000.0; //mm/s 
END_VAR             										
VAR_OUTPUT          										
	ErrorMin												:	BOOL	:= 0;	//Error - IN signal is flickering
	ErrorMax												: 	BOOL	:= 0;	//Error - IN signal is to long TRUE, a sign for jammed material
	TimeInFree												:	TIME	:= T#0MS;
	TimeInOccupied											:	TIME	:= T#0MS;                                                                                                       
END_VAR             	
VAR                 	
	TON_ToMin 												: 	TON;
	TON_ToMax 												: 	TON;
	MemSysTime												:	TIME;
	Mem														:	BYTE := 0;
	CntToMin												:	BYTE	:= 0;
END_VAR

(* monitors the toggle-signal of a sensor		 				       	 V2.2		*)
(************************************************************************************)

(* abort if not enable ***********************************************)
IF NOT Enable	
	OR ErrorMin
	OR ErrorMax
THEN
	Mem.1													:= TRUE;
	IF ResetTrig 
	THEN 
		reset();	
	END_IF
	RETURN;
END_IF
	
(* runtime meassuring *************************************)
TON_ToMin(
	IN 	:= TRUE, 
	PT 	:= LREAL_TO_TIME( ((LenghtMin + Offset_mm) / MAX(1.0, ABS(Velo)) ) * 1000.0) + Offset_msec,
	Q	=> );
	
IF IN AND NOT Mem.0 
THEN
	IF NOT TON_ToMin.Q
	THEN
		CntToMin											:= CntToMin + 1;
	ELSE                                                    	
		CntToMin											:= 0;
	END_IF                                                  	
	ErrorMin												:= CntToMin >= 3;
	TON_ToMin(IN := FALSE);
	TimeInOccupied := T#0MS;
ELSIF NOT In AND Mem.0 
THEN	
	IF NOT TON_ToMin.Q
	THEN
		CntToMin											:= CntToMin + 1;
	ELSE
		CntToMin											:= 0;
	END_IF
	ErrorMin												:= CntToMin >= 3;
	TON_ToMin(IN := FALSE);
	TimeInFree := T#0MS;
END_IF
Mem.0														:= In;

(* runtime error ********************************)
TON_ToMax(
	IN 	:= In AND NOT Mem.1, 
	PT 	:= LREAL_TO_TIME( ((LenghtMax + Offset_mm) / MAX(1.0, ABS(Velo)) ) * 1000.0) + Offset_msec,
	Q	=> ErrorMax);

(* runtime meassuring **************************************************)	
IF Mem.1 
THEN 
	MemSysTime 												:= TIME(); 
END_IF

IF IN 
THEN 
	TimeInOccupied 											:= TimeInOccupied + (TIME() - MemSysTime);
ELSE
	TimeInFree 												:= TimeInFree + (TIME() - MemSysTime);
END_IF
MemSysTime													:= TIME();

(* reset restart ************************************)
Mem.1														:= FALSE;
(********************************************************************************)

METHOD PUBLIC reset : BOOL
VAR_INPUT
END_VAR
ErrorMin := ErrorMAx 								:= FALSE; 
reset												:= TRUE;
END_METHOD

END_FUNCTION_BLOCK

// POUs/TimeHelper/systemtimeCmp
{attribute 'no_check'}
// This Funktionblock compares two Systemtime timestructs datatype with diffrent Options
// Q := In1 = In2 		in dependence of chosen Options
FUNCTION_BLOCK systemtimeCmp
VAR_OUTPUT CONSTANT
{attribute 'displaymode':='binary'}                     	                   
	OPTION_COMPARE_ALL										:	BYTE  := 2#1111_1111;	
{attribute 'displaymode':='binary'}
	OPTION_COMPARE_MS										:	BYTE  := 2#0000_0001;	// Milliseconds
{attribute 'displaymode':='binary'}                                            
	OPTION_COMPARE_S										:	BYTE  := 2#0000_0010;	// Seconds
{attribute 'displaymode':='binary'}                                            
	OPTION_COMPARE_MIN										:	BYTE  := 2#0000_0100;	// Minutes
{attribute 'displaymode':='binary'}                     	                   
	OPTION_COMPARE_H										:	BYTE  := 2#0000_1000;	// Hours
{attribute 'displaymode':='binary'}                     	                   
	OPTION_COMPARE_D										:	BYTE  := 2#0001_0000;	// Days
{attribute 'displaymode':='binary'}                     	                   
	OPTION_COMPARE_DOW										:	BYTE  := 2#0010_0000;	// DayOfWeek
{attribute 'displaymode':='binary'}                     	                   
	OPTION_COMPARE_M										:	BYTE  := 2#0100_0000;	// Months
{attribute 'displaymode':='binary'}                     	                   
	OPTION_COMPARE_Y										:	BYTE  := 2#1000_0000;	// Years
END_VAR
VAR_INPUT
	In1														:	Timestruct;
	In2														:	Timestruct;
	{attribute 'displaymode':='binary'} 
	Options													:	BYTE;		// .0 = ms 
																			// .1 = s 
																			// .2 = min 
																			// .3 = h 
																			// .4 = d 
																			// .5 = dow 
																			// .6 = M 
																			// .7 = Y
END_VAR
VAR_OUTPUT
	Q														:	BOOL;
	Q_RT													:	BOOL;
	Q_FT													:	BOOL;
END_VAR
VAR
END_VAR

			
(***********************************************************)
IF NOT Q THEN
	Q														:=  (Milliseconds(In1,In2) 	OR NOT Options.0)
																AND (Seconds(In1,In2)		OR NOT Options.1)
																AND (Minutes(In1,In2)		OR NOT Options.2)
																AND (Hours(In1,In2)			OR NOT Options.3)
																AND (Days(In1,In2)			OR NOT Options.4)
																AND (DayOfWeek(In1,In2)		OR NOT Options.5)
																AND (Months(In1,In2)		OR NOT Options.6)
																AND (Years(In1,In2)			OR NOT Options.7);
	Q_RT 													:= Q;
	Q_FT 													:= FALSE;
ELSE
	Q														:=  (Milliseconds(In1,In2) 	OR NOT Options.0)
																AND (Seconds(In1,In2)		OR NOT Options.1)
																AND (Minutes(In1,In2)		OR NOT Options.2)
																AND (Hours(In1,In2)			OR NOT Options.3)
																AND (Days(In1,In2)			OR NOT Options.4)
																AND (DayOfWeek(In1,In2)		OR NOT Options.5)
																AND (Months(In1,In2)		OR NOT Options.6)
																AND (Years(In1,In2)			OR NOT Options.7);
	Q_RT 													:= FALSE;
	Q_FT 													:= NOT Q;
END_IF
(***********************************************************)

// returns true if In1.wDayOfWeek = In2.wDayOfWeek
METHOD public dayOfWeek : BOOL
VAR_INPUT
	In1				: TIMESTRUCT;
	In2				: TIMESTRUCT;
END_VAR
DayOfWeek 			:= In1.wDayOfWeek = In2.wDayOfWeek;
END_METHOD

// returns true if In1.wDay = In2.wDay
METHOD PUBLIC days : BOOL
VAR_INPUT
	In1				: TIMESTRUCT;
	In2				: TIMESTRUCT;
END_VAR
Days 				:= In1.wDay = In2.wDay;
END_METHOD

// returns true if In1.wHour = In2.wHour
METHOD public hours : BOOL
VAR_INPUT
	In1				: TIMESTRUCT;
	In2				: TIMESTRUCT;
END_VAR
Hours 				:= In1.wHour = In2.wHour;
END_METHOD

// returns true if In1.wMilliseconds = In2.wMilliseconds
METHOD PUBLIC milliseconds : BOOL
VAR_INPUT
	In1				: TIMESTRUCT;
	In2				: TIMESTRUCT;
END_VAR
Milliseconds 		:= In1.wMilliseconds = In1.wMilliseconds;
END_METHOD

// returns true if In1.wMinute = In2.wMinute
METHOD PUBLIC minutes : BOOL
VAR_INPUT
	In1				: TIMESTRUCT;
	In2				: TIMESTRUCT;
END_VAR
Minutes 			:= In1.wMinute = In2.wMinute;
END_METHOD

// returns true if In1.wMonth = In2.wMonth
METHOD PUBLIC months : BOOL
VAR_INPUT
	In1				: TIMESTRUCT;
	In2				: TIMESTRUCT;
END_VAR
Months				:= In1.wMonth = In2.wMonth;
END_METHOD

// returns true if In1.wSecond = In2.wSecond
METHOD PUBLIC seconds : BOOL
VAR_INPUT
	In1				: TIMESTRUCT;
	In2				: TIMESTRUCT;
END_VAR
Seconds 			:= In1.wSecond = In2.wSecond;
END_METHOD

// returns true if In1.wYear = In2.wYear
METHOD public years : BOOL
VAR_INPUT
	In1			: TIMESTRUCT;
	In2			: TIMESTRUCT;
END_VAR
Years 			:= In1.wYear = In2.wYear;
END_METHOD

END_FUNCTION_BLOCK

// POUs/TimeHelper/systemtimeInCam
{attribute 'no_check'}
// retuns True if In Timestruct is in setpoint +/- window 
// Year and DayOfWeek will except of this comparison 
FUNCTION systemtimeInCam : Bool
VAR_IN_OUT
	In				: TIMESTRUCT;
	SETP			: TIMESTRUCT;
	WINDOW			: TIMESTRUCT;
END_VAR
VAR
	Neg 			: 	WORD;	
	Pos 			:	WORD;
END_VAR

systemtimeInCam			:= FALSE;	

//Neg 				:= TO_WORD(LIMIT(0,TO_INT(SETP.wYear) - TO_INT(WINDOW.wYear),2070));
//Pos 				:= TO_WORD(LIMIT(0,TO_INT(SETP.wYear) + TO_INT(WINDOW.wYear),2070));
//IF 		In.wYear > Neg
//	AND	In.wYear < Pos
//THEN // Year OK
//	IF 		In.wYear = Neg
//		OR	In.wYear = Pos
//	THEN // Year Limit
		Neg 			:= TO_WORD(LIMIT(0,TO_INT(SETP.wMonth) - TO_INT(WINDOW.wMonth),12));
		Pos 			:= TO_WORD(LIMIT(0,TO_INT(SETP.wMonth) + TO_INT(WINDOW.wMonth),12));
		IF 		In.wMonth >= Neg
			AND In.wMonth <= Pos
		THEN // Month OK
			IF 		In.wMonth = Neg
				OR 	In.wMonth = Pos
			THEN // Month Limit
				Neg 			:= TO_WORD(LIMIT(0,TO_INT(SETP.wDay) - TO_INT(WINDOW.wDay),31));
				Pos 			:= TO_WORD(LIMIT(0,TO_INT(SETP.wDay) + TO_INT(WINDOW.wDay),31));
				IF 		In.wDay >= Neg
					AND	In.wDay <= Pos
				THEN // Day OK
					IF 		In.wDay = Neg
						OR	In.wDay = Pos
					THEN // Day Limit
//						Neg 			:= TO_WORD(LIMIT(0,TO_INT(SETP.wDayOfWeek) - TO_INT(WINDOW.wDayOfWeek),7));
//						Pos 			:= TO_WORD(LIMIT(0,TO_INT(SETP.wDayOfWeek) + TO_INT(WINDOW.wDayOfWeek),7));
//						IF 		In.wDayOfWeek >= Neg
//							AND In.wDayOfWeek <= Pos
//						THEN // Dow OK
//							IF 		In.wDayOfWeek = Neg
//								OR	In.wDayOfWeek = Pos
//							THEN // Dow Limit
								Neg 			:= TO_WORD(LIMIT(0,TO_INT(SETP.wHour) - TO_INT(WINDOW.wHour),23));
								Pos 			:= TO_WORD(LIMIT(0,TO_INT(SETP.wHour) + TO_INT(WINDOW.wHour),23));
								IF 		In.wHour >= Neg
									AND	In.wHour <= Pos
								THEN // Hour OK
									IF 		In.wHour = Neg
										OR	In.wHour = Pos
									THEN // Hour Limit
										Neg 			:= TO_WORD(LIMIT(0,TO_INT(SETP.wMinute) - TO_INT(WINDOW.wMinute),60));
										Pos 			:= TO_WORD(LIMIT(0,TO_INT(SETP.wMinute) + TO_INT(WINDOW.wMinute),60));
										IF 		In.wMinute >= Neg
											AND In.wMinute <= Pos
										THEN // Minute OK
											IF		In.wMinute = Neg
												OR	In.wMinute = Pos
											THEN // Minute Limit
												Neg 			:= TO_WORD(LIMIT(0,TO_INT(SETP.wSecond) - TO_INT(WINDOW.wSecond),60));
												Pos 			:= TO_WORD(LIMIT(0,TO_INT(SETP.wSecond) + TO_INT(WINDOW.wSecond),60));
												IF 		In.wSecond >= Neg
													AND	In.wSecond <= Pos
												THEN // Second OK
													IF 		In.wSecond = Neg
														OR	In.wSecond = Pos
													THEN // Second Limit
														Neg 					:= TO_WORD(LIMIT(0,TO_INT(SETP.wMilliseconds) - TO_INT(WINDOW.wMilliseconds),1000));
														Pos 					:= TO_WORD(LIMIT(0,TO_INT(SETP.wMilliseconds) + TO_INT(WINDOW.wMilliseconds),1000));
														IF 		In.wMilliseconds >= Neg
															AND In.wMilliseconds <= Pos
														THEN // Millisecond OK
															systemtimeInCam					:= TRUE;																													
														END_IF	
													ELSE // Second OK
														systemtimeInCam					:= TRUE;
													END_IF
												END_IF
											ELSE // Minute OK
												systemtimeInCam					:= TRUE;
											END_IF
										END_IF
									ELSE // Hour OK
										systemtimeInCam					:= TRUE;
									END_IF
								END_IF
//							ELSE // DOW OK
//								TimestructCAM					:= TRUE;
//							END_IF
//						END_IF
					ELSE // Day OK
						systemtimeInCam					:= TRUE;			
					END_IF
				END_IF
			ELSE // Month OK
				systemtimeInCam					:= TRUE;			
			END_IF
		END_IF 
//	ELSE // Year OK
//		TimestructCAM					:= TRUE;	
//	END_IF	
//END_IF

END_FUNCTION

// POUs/TimeHelper/systemtimeInWin
{attribute 'no_check'}
// retuns True if Low <= In <= High Timestruct datatypes inputs
// 0 value will except part of this comparison
FUNCTION systemtimeInWin : Bool
VAR_IN_OUT
	In														: TIMESTRUCT;
	Low														: TIMESTRUCT;
	High													: TIMESTRUCT;
END_VAR
VAR
	LowOK													: BOOL;
	HighOK													: BOOL;
END_VAR

systemtimeInWin												:= FALSE;
LowOK														:= FALSE;
HighOK														:= FALSE;

IF In.wYear > Low.wYear THEN
	LowOK													:= TRUE;
ELSIF In.wYear = Low.wYear THEN
	IF In.wMonth > Low.wMonth THEN
			LowOK											:= TRUE;
	ELSIF In.wMonth = Low.wMonth THEN
		IF In.wDay > Low.wDay THEN
			LowOK											:= TRUE;
		ELSIF In.wDay = Low.wDay THEN
			IF In.wDayOfWeek > Low.wDayOfWeek THEN
				LowOK										:= TRUE;
			ELSIF In.wDayOfWeek = Low.wDayOfWeek THEN
				IF In.wHour > Low.wHour THEN
					LowOK									:= TRUE;
				ELSIF In.wHour = Low.wHour THEN
					IF In.wMinute > Low.wMinute THEN
						LowOK								:= TRUE;
					ELSIF In.wMinute = Low.wMinute THEN
						IF In.wSecond > Low.wSecond THEN
							LowOK							:= TRUE;
						ELSIF In.wSecond = Low.wSecond THEN
							IF In.wMilliseconds >= Low.wMilliseconds THEN
								LowOK						:= TRUE;
							END_IF	// ms
						END_IF	//s
					END_IF	//min 
				END_IF	// h
			END_IF	// dow
		END_IF	// d
	END_IF	// M
END_IF	// Y

IF In.wYear < High.wYear THEN
	HighOK													:= TRUE;
ELSIF In.wYear = High.wYear
	OR_ELSE High.wYear = 0
THEN
	IF In.wMonth < High.wMonth THEN
			HighOK											:= TRUE;
	ELSIF In.wMonth = High.wMonth
		 OR_ELSE High.wMonth = 0
	THEN
		IF In.wDay < High.wDay THEN
			HighOK											:= TRUE;
		ELSIF In.wDay = High.wDay 
			OR_ELSE High.wDay = 0
		THEN
			IF In.wDayOfWeek < High.wDayOfWeek THEN
				HighOK										:= TRUE;
			ELSIF In.wDayOfWeek = High.wDayOfWeek 
				OR_ELSE High.wDayOfWeek = 0
			THEN
				IF In.wHour < High.wHour THEN
					HighOK									:= TRUE;
				ELSIF In.wHour = High.wHour 
					OR_ELSE High.wHour = 0
				THEN
					IF In.wMinute < High.wMinute THEN
						HighOK								:= TRUE;
					ELSIF In.wMinute = High.wMinute 
						OR_ELSE High.wMinute = 0
					THEN
						IF In.wSecond < High.wSecond THEN
							HighOK							:= TRUE;
						ELSIF In.wSecond = High.wSecond 
							OR_ELSE High.wSecond = 0
						THEN
							IF In.wMilliseconds <= High.wMilliseconds 
								OR_ELSE High.wMilliseconds = 0
							THEN
								HighOK						:= TRUE;
							END_IF	// ms
						END_IF	//s
					END_IF	//min 
				END_IF	// h
			END_IF	// dow
		END_IF	// d
	END_IF	// M
END_IF	// Y

systemtimeInWin												:= LowOK AND HighOK;

END_FUNCTION

// POUs/TimeHelper/TimeSwitch
{attribute 'no_check'}
//Simpel single time switch based on actual date and time, configured by time of day values for on and off
FUNCTION_BLOCK TimeSwitch
VAR_INPUT
	 Enable                                  				:  	BOOL;			//Start time switch - FALSE = set Q back to FALSE
	 ActDT			                          				:	DATE_AND_TIME;	//Actual date and time
	 SwitchOnTOD                             				: 	TOD;			//Time of day where Q will set to TRUE 
	 SwitchOffTOD                            				:  	TOD;			//Time of day where Q will set back to FALSE 
{attribute 'displaymode':='binary'}
	 DayConfig												:	BYTE := 2#0000_0000;//.0 = Sun|.1 = Mon|.2 = Tue|.3 = Wed|.4 = Thu|.5 = Fri|.6 = Sat|.7 = full week																							
END_VAR                                                 	
VAR_OUTPUT
	 Q                                       				 :  BOOL;			//Output is TRUE between SwitchOnTOD and SwitchOFfTOD
	 Q_RT                                    				 :  BOOL;			//Rising flag of Q
	 Q_FT                                    				 :  BOOL;			//Falling flag of Q
END_VAR
VAR
	 tmpCTS                                   				:  TIMESTRUCT;
	 tmpActTOD                            					:  TOD;
	 MemQ													:	BOOL;
END_VAR

IF Enable 
	AND ActDT > DT#1970-01-01-00:00
	AND ActDT < DT#2106-02-06-06:28:15
THEN
	tmpCTS 													:= DT_TO_SYSTEMTIME(ActDT);
	tmpActTOD 												:= DT_TO_TOD(ActDT);
	IF SwitchOnTOD < SwitchOffTOD 
	THEN
		MemQ												:= Q;
		IF tmpActTOD >= SwitchOnTOD 
			AND tmpActTOD < SwitchOffTOD
 		THEN			
			Q												:= tmpCTS.wDayOfWeek = 0 AND DayConfig.0 //Sunday
																OR tmpCTS.wDayOfWeek = 1 AND DayConfig.1
																OR tmpCTS.wDayOfWeek = 2 AND DayConfig.2
																OR tmpCTS.wDayOfWeek = 3 AND DayConfig.3
																OR tmpCTS.wDayOfWeek = 4 AND DayConfig.4
																OR tmpCTS.wDayOfWeek = 5 AND DayConfig.5
																OR tmpCTS.wDayOfWeek = 6 AND DayConfig.6 //Saturday
																OR DayConfig.7;
                    										
		ELSE        	
			Q												:= FALSE;			
		END_IF      										
		Q_RT												:= Q AND NOT MemQ;
		Q_FT												:= NOT Q AND MemQ;

	ELSIF SwitchOnTOD > SwitchOffTOD
	THEN 
		MemQ												:= Q;
		IF tmpActTOD >= SwitchOnTOD 
		THEN
			Q												:= tmpCTS.wDayOfWeek = 0 AND DayConfig.0 //Sunday
																OR tmpCTS.wDayOfWeek = 1 AND DayConfig.1
																OR tmpCTS.wDayOfWeek = 2 AND DayConfig.2
																OR tmpCTS.wDayOfWeek = 3 AND DayConfig.3
																OR tmpCTS.wDayOfWeek = 4 AND DayConfig.4
																OR tmpCTS.wDayOfWeek = 5 AND DayConfig.5
																OR tmpCTS.wDayOfWeek = 6 AND DayConfig.6 //Saturday
																OR DayConfig.7;
		
		ELSIF tmpActTOD < SwitchOnTOD 
			AND tmpActTOD >= SwitchOffTOD 
		THEN
			Q 												:= FALSE;
		END_IF      										
		Q_RT												:= Q AND NOT MemQ;
		Q_FT												:= NOT Q AND MemQ;
	END_IF          										
ELSE	            										
	Q														:= FALSE;
	Q_RT													:= FALSE;
	Q_FT													:= FALSE;
END_IF

END_FUNCTION_BLOCK

// POUs/TimeHelper/TONRecord
{attribute 'no_check'}
//TON with the possibility to accumulate the time value
FUNCTION_BLOCK TONRecord
VAR_INPUT
	IN														: BOOL := FALSE;//Start time accumulation
	ResetTrig												: BOOL := FALSE;//Reset function block
	PT														: TIME := T#0MS;//time to pass, before Q is set TRUE
	OFFSET													: TIME := T#0MS;//Start time offset 
END_VAR                             						
VAR_OUTPUT                          						
	Q														: BOOL := FALSE;//TRUE if time is passed 
	ET														: TIME;			//Elapsed time
END_VAR                             						
VAR                                 	
	state													: INT := 0;
	TimeDP2													: TON;
	elapsedTime												: TIME;
END_VAR

IF ResetTrig THEN
	reset();
ELSE
	CASE state OF
	0: //Wait for start timer
		Q	 												:= FALSE;
		IF IN THEN
			elapsedTime 									:= T#0MS + OFFSET;
			ET 												:= elapsedTime;
			TimeDP2(IN := FALSE);
			TimeDP2(IN := TRUE, PT := PT-elapsedTime);
			State 											:= 20;
		END_IF
	20: //Run timer
		TimeDP2();
		ET 													:= elapsedTime + TimeDP2.ET;
		IF NOT IN 
		THEN
			state 											:= 30;
		ELSIF TimeDP2.q 
		THEN
			Q	 											:= TRUE;
			state 											:= 99;
		END_IF
	30: //Restart timer
		IF IN 
		THEN
			IF PT >= elapsedTime 
			THEN 
				TimeDP2(IN := FALSE);
				TimeDP2(IN := TRUE, PT := PT-elapsedTime);
				state 										:= 20;
			ELSE        									
				Q	 										:= TRUE;
				state 										:= 99;
			END_IF
		END_IF
	END_CASE
END_IF

METHOD PUBLIC reset : booL //Return value = TRUE if execution finished
VAR_INPUT
END_VAR
elapsedTime 												:= T#0MS + OFFSET;
ET 															:= elapsedTime;
TimeDP2(IN := FALSE);
state 														:= 0;
Q															:= FALSE;
reset														:= TRUE;
END_METHOD

END_FUNCTION_BLOCK

// POUs/TimeHelper/TONTOF
{attribute 'no_check'}
//Timer with on off-delay
FUNCTION_BLOCK TONTOF
VAR_INPUT
	IN														:	BOOL := FALSE; //Return value TRUE = starts delay on (TON), FALSE starts delay of in case output Q is TRUE
	RST														:	BOOL := FALSE; //Reset timer and set Q to false
	PT_ON													:	TIME := T#0MS; //time to pass, before Q is set TRUE
	PT_OFF													:	TIME := T#0MS; //time to pass, before Q is set back to FALSE
END_VAR         											
VAR_OUTPUT      											
	Q														:	BOOL := FALSE;//TRUE if time is passed 
END_VAR         											
VAR             	
	TON														:	TON;
END_VAR

IF RST
THEN
	reset();
ELSIF NOT Q 
THEN
	TON(IN := IN, PT := PT_ON , Q => Q);
	IF Q 
	THEN 
		TON(IN := FALSE); 
	END_IF
ELSE
	TON(IN := NOT IN, PT := PT_OFF);
	Q := NOT TON.Q;
	IF NOT Q 
	THEN 
		TON(IN := FALSE); 
	END_IF
END_IF

{attribute 'monitoring' := 'call'}
PROPERTY PUBLIC BT : TIME
GET
IF ton.IN
	AND NOT ton.Q
THEN
	BT 														:= ton.PT - ton.ET;
ELSE       													
	BT 														:= T#0MS;
END_IF
END_GET
END_PROPERTY

METHOD PUBLIC reset : BOOL //Return value = TRUE if execution finished
VAR_INPUT
END_VAR
Q 															:= FALSE;
TON(IN := FALSE);
reset													:= TRUE;
END_METHOD

END_FUNCTION_BLOCK

// POUs/TimeHelper/VeloLinearMeasurement
{attribute 'no_check'}
//Accumulates the covered distance based on the velocity input and the time IN is TRUE - used to detect jamped pieces on a conveyor
FUNCTION_BLOCK VeloLinearMeasurement
VAR_INPUT
	Enable													:	BOOL;	//Enable function (e.g. Conveyor on)
	ResetTrig												:	BOOL;	//Reset Q
	IN														:	BOOL; 	//Sensor input
	Velo													:	LREAL;  //mm/ms | m/s with FACTOR=1, m/min with FACTOR=16.666666666666668
	Factor													:	LREAL := 1.0;	//Used to convert "VELO" into mm/ms (e.g. 16.666666666666668 to convert m/min into mm/ms
END_VAR             										
VAR_OUTPUT          										
	Q														:	LREAL;	//Accumulated value in mm
END_VAR             										
VAR                 										
	tx														:	DWORD;
	last 													: 	DWORD;
	ms														: 	DWORD;
	mmProms													:	LREAL;
END_VAR


(* Get mm pro ms *)
mmProms 													:= VELO * FACTOR; 

(* read system time *)
tx 															:= TIME_TO_DWORD(TIME());

(* Sequence *)
IF ResetTrig THEN
	reset();
ELSIF IN AND Enable THEN
	(* add the current milliseconds *)
	ms 														:= (tx - last) + ms;
	Q 														:= ms * mmProms;
ELSE
	;
END_IF

(* Save last Cylcetime *)
last 														:= tx;

(**********************************************************************)

METHOD PUBLIC reset : bool //Return value = TRUE if execution finished
VAR_INPUT
END_VAR
Q 															:= 0;
ms 															:= 0;
reset													:= TRUE;
END_METHOD

END_FUNCTION_BLOCK

// Version/disclaimerStatement
// .. Disclaimer:: This function contains statements about the use of this library 
{attribute 'no-analysis'}
{attribute 'no_check'}
FUNCTION disclaimerStatement : WSTRING(1500)
VAR_INPUT
END_VAR
VAR
END_VAR

DisclaimerStatement := 
	"This disclaimer contains statements about the use of this library.

		-The use of this version of the library is free of charge 
		-It is incumbent on the customer to check and decide whether the library and provided function is suitable for use his particular application
		-This library is provided 'AS IS' and neither a part of TwinCAT3 nor directly supported by Beckhoff Automation
		-The use of the Library is at the Customer's own risk
		-There is no warranty given that the library and source code, which is made available with this library is complete or accurate
		-In no event will the author or Beckhoff Automation be liable for any claims, damages or other liability for errors and/or omissions arising from the use of the library
		-There is no right to expect maintenance, support, enhancements or modifications of the library as well as for updates or compatibility to updates of the library or TwinCAT3 if released
		
	For feedback or questions please contact the Beckhoff Industry Management for Electronics Manufacturing, D.Schlingmann@Beckhoff.com
	
	© Beckhoff Automation GmbH & Co. KG,
	The reproduction, distribution and utilisation of this library or parts of it as well as the communication of its content to others without express authorisation is prohibited held liable for the payment of damages.
	
	All rights reserved in the event of the grant of a patent, utility model or design.";

END_FUNCTION
